// TIA Portal V18 export
DATA_BLOCK "SS2_A4_32DO_DO_Vars"   // DB11151
{ S7_Optimized_Access := 'FALSE' }
VERSION : 0.1
// stored: AutoNumber false, DBAccessibleFromOPCUA true, IsOnlyStoredInLoadMemory false, IsWriteProtectedInAS false
   VAR
      DO1 { S7_SetPoint := 'True'} : "UDT_DOadv";
      DO2 { S7_SetPoint := 'True'} : "UDT_DOadv";
      DO3 { S7_SetPoint := 'True'} : "UDT_DOadv";
      DO4 : "UDT_DOadv";
      DO5 { S7_SetPoint := 'True'} : "UDT_DOadv";
      DO6 { S7_SetPoint := 'True'} : "UDT_DOadv";
      DO7 { S7_SetPoint := 'True'} : "UDT_DOadv";
      DO8 { S7_SetPoint := 'True'} : "UDT_DOadv";
      DO9 { S7_SetPoint := 'True'} : "UDT_DOadv";
      DO10 { S7_SetPoint := 'True'} : "UDT_DOadv";
      DO11 { S7_SetPoint := 'True'} : "UDT_DOadv";
      DO12 { S7_SetPoint := 'True'} : "UDT_DOadv";
      DO13 { S7_SetPoint := 'True'} : "UDT_DOadv";
      DO14 { S7_SetPoint := 'True'} : "UDT_DOadv";
      DO15 { S7_SetPoint := 'True'} : "UDT_DOadv";
      DO16 { S7_SetPoint := 'True'} : "UDT_DOadv";
      DO17 { S7_SetPoint := 'True'} : "UDT_DOadv";
      DO18 { S7_SetPoint := 'True'} : "UDT_DOadv";
      DO19 { S7_SetPoint := 'True'} : "UDT_DOadv";
      DO20 { S7_SetPoint := 'True'} : "UDT_DOadv";
      DO21 { S7_SetPoint := 'True'} : "UDT_DOadv";
      DO22 { S7_SetPoint := 'True'} : "UDT_DOadv";
      DO23 { S7_SetPoint := 'True'} : "UDT_DOadv";
      DO24 { S7_SetPoint := 'True'} : "UDT_DOadv";
      DO25 { S7_SetPoint := 'True'} : "UDT_DOadv";
      DO26 { S7_SetPoint := 'True'} : "UDT_DOadv";
      DO27 { S7_SetPoint := 'True'} : "UDT_DOadv";
      DO28 { S7_SetPoint := 'True'} : "UDT_DOadv";
      DO29 { S7_SetPoint := 'True'} : "UDT_DOadv";
      DO30 { S7_SetPoint := 'True'} : "UDT_DOadv";
      DO31 { S7_SetPoint := 'True'} : "UDT_DOadv";
      DO32 { S7_SetPoint := 'True'} : "UDT_DOadv";
   END_VAR
BEGIN
   DO2.iFuncSystemID := 2;
   DO2.iFuncVar := 1;
   DO3.iFuncSystemID := 2;
   DO4.iFuncSystemID := 2;
   DO4.iFuncVar := 3;
   DO5.iFuncSystemID := 10;
   DO5.iFuncVar := 17;
   DO6.iFuncSystemID := 10;
   DO6.iFuncVar := 18;
   DO7.iFuncSystemID := 10;
   DO7.iFuncVar := 7;
   DO8.iFuncSystemID := 10;
   DO8.iFuncVar := 8;
   DO9.iFuncSystemID := 10;
   DO9.iFuncVar := 19;
   DO13.iFuncSystemID := 10;
   DO13.iFuncVar := 16;
END_DATA_BLOCK
